(* IEC 61131-3 sources: KrizikProgramovani/Mosaic/TecoApp/Kriz/PocetKroku, 1 file *)

(* ---- POCETKROKU.ST ---- *)
VAR_GLOBAL
  hodnota : INT;
END_VAR
